(* CoDeSys 2.3.9.41 project: TASK_PRIO.pro *)
(* Libraries: STANDARD.LIB 5.6.98 11:03:02 *)

(* Task configuration *)
TASK MAIN1 (PRIORITY := 2, INTERVAL := T#200ms);
	MAIN1();
END_TASK
TASK MAIN2 (PRIORITY := 1, INTERVAL := T#120ms);
	MAIN2();
END_TASK
TASK MAIN3 (PRIORITY := 0, INTERVAL := T#100ms);
	MAIN3();
END_TASK

(* POU MAIN1, ST *)
PROGRAM MAIN1
VAR
END_VAR
;
END_PROGRAM

(* POU MAIN2, ST *)
PROGRAM MAIN2
VAR
END_VAR
;
END_PROGRAM

(* POU MAIN3, ST *)
PROGRAM MAIN3
VAR
END_VAR
;
END_PROGRAM
